// TIA Portal V18 export
// export: Created 2025-12-01T12:38:49.4516344Z, ExportSetting None, DisplayName Totally Integrated Automation Portal, DisplayVersion V18 Update 5, DisplayName TIA Portal Openness, DisplayVersion V18 Update 5, DisplayName TIA Portal Teamcenter Gateway, DisplayVersion V18, DisplayName TIA Portal Version Control Interface, DisplayVersion V18, DisplayName STEP 7 Professional, DisplayVersion V18 Update 5, DisplayName STEP 7 Safety, DisplayVersion V18, DisplayName WinCC Professional, DisplayVersion V18 Update 5
FUNCTION "Gluing" : Void   // FC2800, LAD
{ S7_Optimized_Access := 'TRUE' }
// stored: AutoNumber false, SetENOAutomatically false
   VAR_TEMP   // added for the SCL form of the ladder/FBD networks
      _w1 : Bool;
      _w2 : Bool;
   END_VAR
BEGIN

REGION Network 1 (SCL): Input and Output
   //   Input
   "GluingControl".Input.GluingDeviceReady := "iC- GluingDeviceReady";
   "GluingControl".Input.GluingFault := "iC- GluingFault";
   "GluingControl".Input.GluingRefillTank := "iC- GluingRefillTank";
   "GluingControl".Input.GluingTankEmpty := "iC- GluingTankEmpty";

   //   Output
   "oC-GluingPro_X" := "GluingControl".Output.GluingPro_X;
   "oC-GluingPro_Y" := "GluingControl".Output.GluingPro_Y;
   "oC-GluingPro_Z" := "GluingControl".Output.GluingPro_Z;
   "oC-GluingReset" := "GluingControl".Output.GluingReset;
END_REGION

REGION Network 2: Reset
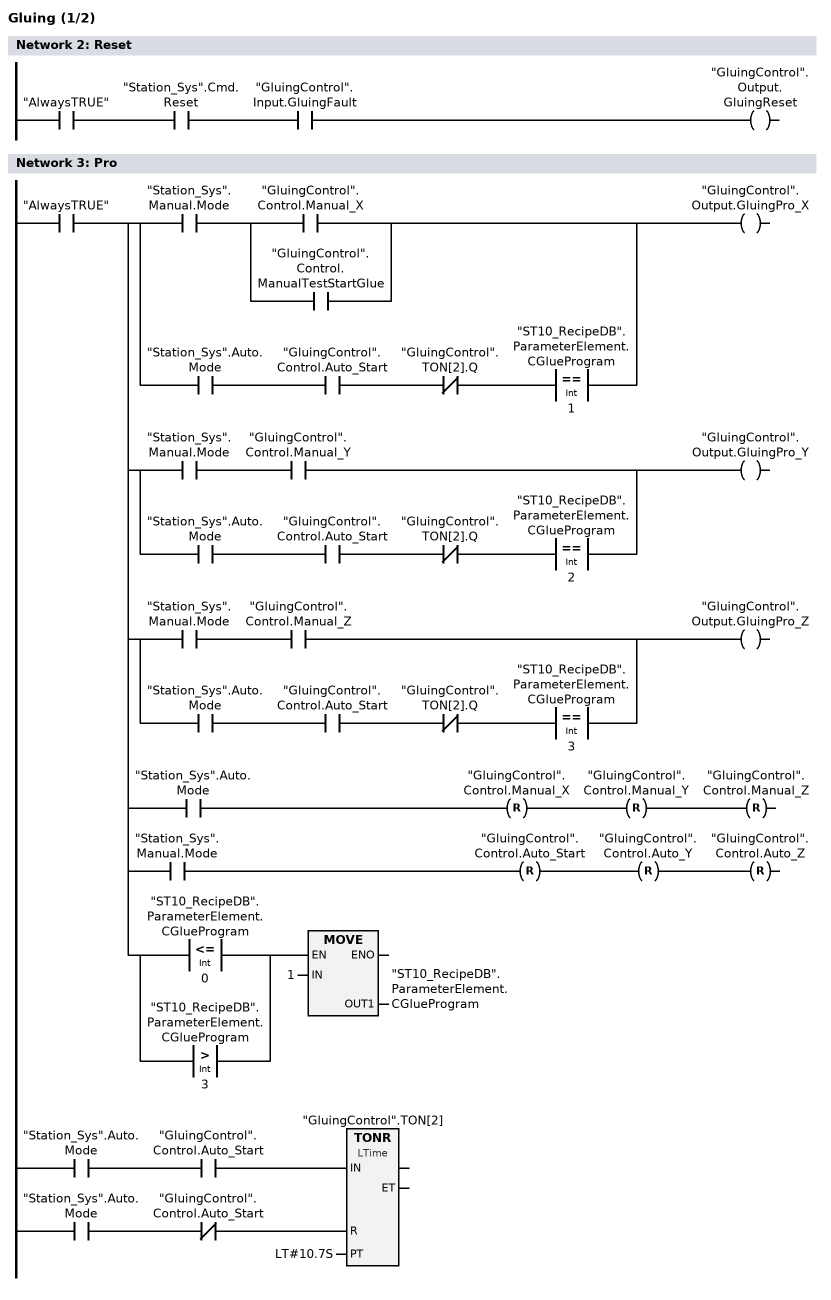
   RUNG wire#powerrail
      Contact( "AlwaysTRUE" )
      Contact( "Station_Sys".Cmd.Reset )
      Contact( "GluingControl".Input.GluingFault )
      Coil( "GluingControl".Output.GluingReset )
   END_RUNG
   // the same network as SCL:
   "GluingControl".Output.GluingReset := "AlwaysTRUE" AND "Station_Sys".Cmd.Reset AND "GluingControl".Input.GluingFault;
END_REGION

REGION Network 3: Pro
   RUNG wire#powerrail
      Contact( "AlwaysTRUE" )
      wire#w1
      Contact( "Station_Sys".Manual.Mode )
      wire#w2
      Contact( "GluingControl".Control.Manual_X )
      wire#w3
      Coil( "GluingControl".Output.GluingPro_X )
   END_RUNG
   RUNG wire#w2
      Contact( "GluingControl".Control.ManualTestStartGlue )
   END_RUNG wire#w3
   RUNG wire#w1
      Contact( "Station_Sys".Auto.Mode )
      Contact( "GluingControl".Control.Auto_Start )
      I_Contact( "GluingControl".TON[2].Q )
      { S7_Templates := "SrcType := Int" } EQ_Contact(in1 := "ST10_RecipeDB".ParameterElement.CGlueProgram, in2 := 1)
   END_RUNG wire#w3
   RUNG wire#w1
      Contact( "Station_Sys".Manual.Mode )
      Contact( "GluingControl".Control.Manual_Y )
      wire#w4
      Coil( "GluingControl".Output.GluingPro_Y )
   END_RUNG
   RUNG wire#w1
      Contact( "Station_Sys".Auto.Mode )
      Contact( "GluingControl".Control.Auto_Start )
      I_Contact( "GluingControl".TON[2].Q )
      { S7_Templates := "SrcType := Int" } EQ_Contact(in1 := "ST10_RecipeDB".ParameterElement.CGlueProgram, in2 := 2)
   END_RUNG wire#w4
   RUNG wire#w1
      Contact( "Station_Sys".Manual.Mode )
      Contact( "GluingControl".Control.Manual_Z )
      wire#w5
      Coil( "GluingControl".Output.GluingPro_Z )
   END_RUNG
   RUNG wire#w1
      Contact( "Station_Sys".Auto.Mode )
      Contact( "GluingControl".Control.Auto_Start )
      I_Contact( "GluingControl".TON[2].Q )
      { S7_Templates := "SrcType := Int" } EQ_Contact(in1 := "ST10_RecipeDB".ParameterElement.CGlueProgram, in2 := 3)
   END_RUNG wire#w5
   RUNG wire#w1
      Contact( "Station_Sys".Auto.Mode )
      R_Coil( "GluingControl".Control.Manual_X )
      R_Coil( "GluingControl".Control.Manual_Y )
      R_Coil( "GluingControl".Control.Manual_Z )
   END_RUNG
   RUNG wire#w1
      Contact( "Station_Sys".Manual.Mode )
      R_Coil( "GluingControl".Control.Auto_Start )
      R_Coil( "GluingControl".Control.Auto_Y )
      R_Coil( "GluingControl".Control.Auto_Z )
   END_RUNG
   RUNG wire#w1
      { S7_Templates := "SrcType := Int" } LE_Contact(in1 := "ST10_RecipeDB".ParameterElement.CGlueProgram, in2 := 0)
      wire#w6
      Move(in := 1, out1 => "ST10_RecipeDB".ParameterElement.CGlueProgram)
   END_RUNG
   RUNG wire#w1
      { S7_Templates := "SrcType := Int" } GT_Contact(in1 := "ST10_RecipeDB".ParameterElement.CGlueProgram, in2 := 3)
   END_RUNG wire#w6
   RUNG wire#powerrail
      Contact( "Station_Sys".Auto.Mode )
      Contact( "GluingControl".Control.Auto_Start )
      { S7_Templates := "time_type := LTime" } "GluingControl".TON[2].TONR(r := wire#w7, pt := LT#10.7S, et =>)
   END_RUNG
   RUNG wire#powerrail
      Contact( "Station_Sys".Auto.Mode )
      I_Contact( "GluingControl".Control.Auto_Start )
   END_RUNG wire#w7
   // the same network as SCL:
   "GluingControl".Output.GluingPro_X := "AlwaysTRUE" AND (("Station_Sys".Manual.Mode AND ("GluingControl".Control.Manual_X OR "GluingControl".Control.ManualTestStartGlue)) OR ("Station_Sys".Auto.Mode AND "GluingControl".Control.Auto_Start AND NOT "GluingControl".TON[2].Q AND ("ST10_RecipeDB".ParameterElement.CGlueProgram = 1)));
   "GluingControl".Output.GluingPro_Y := "AlwaysTRUE" AND (("Station_Sys".Manual.Mode AND "GluingControl".Control.Manual_Y) OR ("Station_Sys".Auto.Mode AND "GluingControl".Control.Auto_Start AND NOT "GluingControl".TON[2].Q AND ("ST10_RecipeDB".ParameterElement.CGlueProgram = 2)));
   "GluingControl".Output.GluingPro_Z := "AlwaysTRUE" AND (("Station_Sys".Manual.Mode AND "GluingControl".Control.Manual_Z) OR ("Station_Sys".Auto.Mode AND "GluingControl".Control.Auto_Start AND NOT "GluingControl".TON[2].Q AND ("ST10_RecipeDB".ParameterElement.CGlueProgram = 3)));
   IF "AlwaysTRUE" AND "Station_Sys".Auto.Mode THEN
       "GluingControl".Control.Manual_X := FALSE;
       "GluingControl".Control.Manual_Y := FALSE;
       "GluingControl".Control.Manual_Z := FALSE;
   END_IF;
   IF "AlwaysTRUE" AND "Station_Sys".Manual.Mode THEN
       "GluingControl".Control.Auto_Start := FALSE;
       "GluingControl".Control.Auto_Y := FALSE;
       "GluingControl".Control.Auto_Z := FALSE;
   END_IF;
   IF "AlwaysTRUE" AND (("ST10_RecipeDB".ParameterElement.CGlueProgram <= 0) OR ("ST10_RecipeDB".ParameterElement.CGlueProgram > 3)) THEN
       "ST10_RecipeDB".ParameterElement.CGlueProgram := 1;
   END_IF;
   "GluingControl".TON[2].TONR(IN := "Station_Sys".Auto.Mode AND "GluingControl".Control.Auto_Start,
                           R := "Station_Sys".Auto.Mode AND NOT "GluingControl".Control.Auto_Start,
                           PT := LT#10.7S);
END_REGION

REGION Network 4: Test
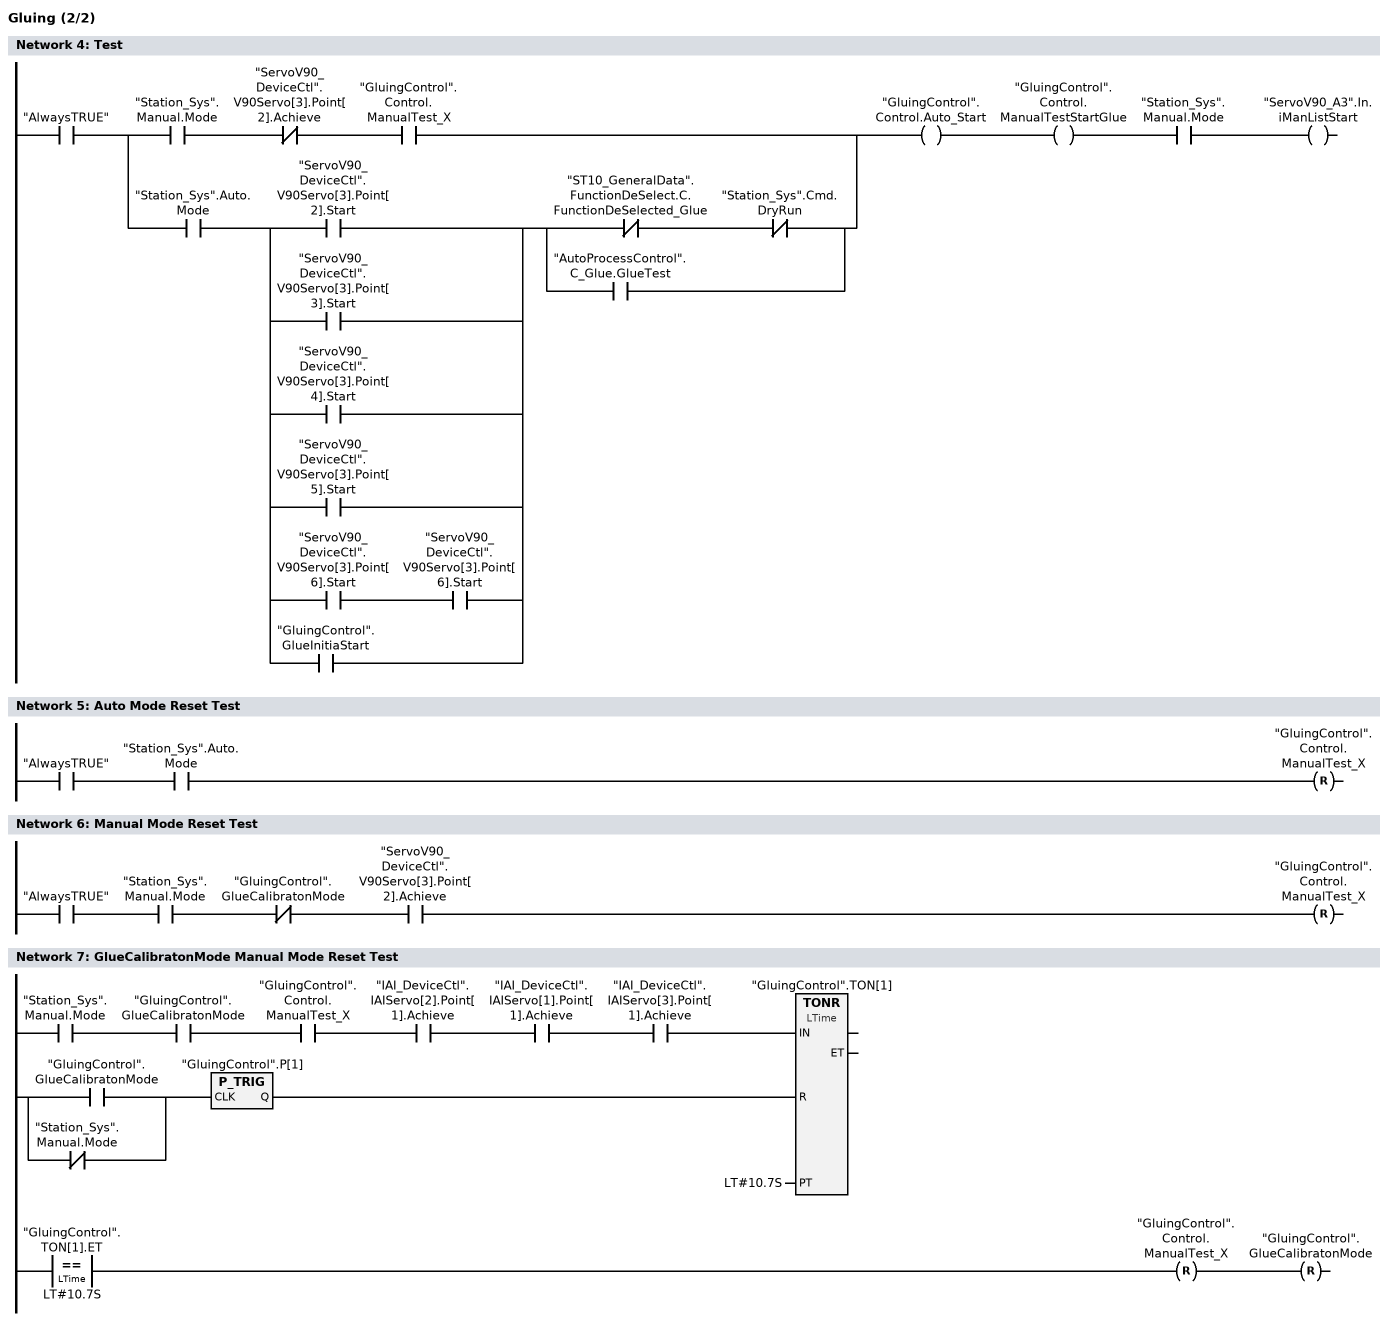
   RUNG wire#powerrail
      Contact( "AlwaysTRUE" )
      wire#w1
      Contact( "Station_Sys".Manual.Mode )
      I_Contact( "ServoV90_DeviceCtl".V90Servo[3].Point[2].Achieve )
      Contact( "GluingControl".Control.ManualTest_X )
      wire#w2
      Coil( "GluingControl".Control.Auto_Start )
      Coil( "GluingControl".Control.ManualTestStartGlue )
      Contact( "Station_Sys".Manual.Mode )
      Coil( "ServoV90_A3".In.iManListStart )
   END_RUNG
   RUNG wire#w1
      Contact( "Station_Sys".Auto.Mode )
      wire#w3
      Contact( "ServoV90_DeviceCtl".V90Servo[3].Point[2].Start )
      wire#w4
      I_Contact( "ST10_GeneralData".FunctionDeSelect.C.FunctionDeSelected_Glue )
      I_Contact( "Station_Sys".Cmd.DryRun )
   END_RUNG wire#w2
   RUNG wire#w3
      Contact( "ServoV90_DeviceCtl".V90Servo[3].Point[3].Start )
   END_RUNG wire#w4
   RUNG wire#w3
      Contact( "ServoV90_DeviceCtl".V90Servo[3].Point[4].Start )
   END_RUNG wire#w4
   RUNG wire#w3
      Contact( "ServoV90_DeviceCtl".V90Servo[3].Point[5].Start )
   END_RUNG wire#w4
   RUNG wire#w3
      Contact( "ServoV90_DeviceCtl".V90Servo[3].Point[6].Start )
      Contact( "ServoV90_DeviceCtl".V90Servo[3].Point[6].Start )
   END_RUNG wire#w4
   RUNG wire#w3
      Contact( "GluingControl".GlueInitiaStart )
   END_RUNG wire#w4
   RUNG wire#w4
      Contact( "AutoProcessControl".C_Glue.GlueTest )
   END_RUNG wire#w2
   // the same network as SCL:
   "GluingControl".Control.Auto_Start := "AlwaysTRUE" AND (("Station_Sys".Manual.Mode AND NOT "ServoV90_DeviceCtl".V90Servo[3].Point[2].Achieve AND "GluingControl".Control.ManualTest_X) OR ("Station_Sys".Auto.Mode AND ("ServoV90_DeviceCtl".V90Servo[3].Point[2].Start OR "ServoV90_DeviceCtl".V90Servo[3].Point[3].Start OR "ServoV90_DeviceCtl".V90Servo[3].Point[4].Start OR "ServoV90_DeviceCtl".V90Servo[3].Point[5].Start OR ("ServoV90_DeviceCtl".V90Servo[3].Point[6].Start AND "ServoV90_DeviceCtl".V90Servo[3].Point[6].Start) OR "GluingControl".GlueInitiaStart) AND ((NOT "ST10_GeneralData".FunctionDeSelect.C.FunctionDeSelected_Glue AND NOT "Station_Sys".Cmd.DryRun) OR "AutoProcessControl".C_Glue.GlueTest)));
   "GluingControl".Control.ManualTestStartGlue := "GluingControl".Control.Auto_Start;
   "ServoV90_A3".In.iManListStart := "GluingControl".Control.Auto_Start AND "Station_Sys".Manual.Mode;
END_REGION

REGION Network 5: Auto Mode Reset Test
   RUNG wire#powerrail
      Contact( "AlwaysTRUE" )
      Contact( "Station_Sys".Auto.Mode )
      R_Coil( "GluingControl".Control.ManualTest_X )
   END_RUNG
   // the same network as SCL:
   IF "AlwaysTRUE" AND "Station_Sys".Auto.Mode THEN "GluingControl".Control.ManualTest_X := FALSE; END_IF;
END_REGION

REGION Network 6: Manual Mode Reset Test
   RUNG wire#powerrail
      Contact( "AlwaysTRUE" )
      Contact( "Station_Sys".Manual.Mode )
      I_Contact( "GluingControl".GlueCalibratonMode )
      Contact( "ServoV90_DeviceCtl".V90Servo[3].Point[2].Achieve )
      R_Coil( "GluingControl".Control.ManualTest_X )
   END_RUNG
   // the same network as SCL:
   IF "AlwaysTRUE" AND "Station_Sys".Manual.Mode AND NOT "GluingControl".GlueCalibratonMode AND "ServoV90_DeviceCtl".V90Servo[3].Point[2].Achieve THEN
       "GluingControl".Control.ManualTest_X := FALSE;
   END_IF;
END_REGION

REGION Network 7: GlueCalibratonMode Manual Mode Reset Test
   RUNG wire#powerrail
      Contact( "Station_Sys".Manual.Mode )
      Contact( "GluingControl".GlueCalibratonMode )
      Contact( "GluingControl".Control.ManualTest_X )
      Contact( "IAI_DeviceCtl".IAIServo[2].Point[1].Achieve )
      Contact( "IAI_DeviceCtl".IAIServo[1].Point[1].Achieve )
      Contact( "IAI_DeviceCtl".IAIServo[3].Point[1].Achieve )
      { S7_Templates := "time_type := LTime" } "GluingControl".TON[1].TONR(r := wire#w2, pt := LT#10.7S, et =>)
   END_RUNG
   RUNG wire#powerrail
      Contact( "GluingControl".GlueCalibratonMode )
      wire#w1
      P_Trig( "GluingControl".P[1] )
   END_RUNG wire#w2
   RUNG wire#powerrail
      I_Contact( "Station_Sys".Manual.Mode )
   END_RUNG wire#w1
   RUNG wire#powerrail
      { S7_Templates := "SrcType := LTime" } EQ_Contact(in1 := "GluingControl".TON[1].ET, in2 := LT#10.7S)
      R_Coil( "GluingControl".Control.ManualTest_X )
      R_Coil( "GluingControl".GlueCalibratonMode )
   END_RUNG
   // the same network as SCL:
   #_w1 := "GluingControl".GlueCalibratonMode OR NOT "Station_Sys".Manual.Mode;
   #_w2 := #_w1 AND NOT "GluingControl".P[1];   // rising edge
   "GluingControl".P[1] := #_w1;
   "GluingControl".TON[1].TONR(IN := "Station_Sys".Manual.Mode AND "GluingControl".GlueCalibratonMode AND "GluingControl".Control.ManualTest_X AND "IAI_DeviceCtl".IAIServo[2].Point[1].Achieve AND "IAI_DeviceCtl".IAIServo[1].Point[1].Achieve AND "IAI_DeviceCtl".IAIServo[3].Point[1].Achieve,
                           R := #_w2,
                           PT := LT#10.7S);
   IF "GluingControl".TON[1].ET = LT#10.7S THEN
       "GluingControl".Control.ManualTest_X := FALSE;
       "GluingControl".GlueCalibratonMode := FALSE;
   END_IF;
END_REGION
END_FUNCTION
